// TIA Portal V20 export
TYPE "LBP_typeModularMcpModeGroupInput"
TITLE = Modular MCP image / Image MCP modulaire
// Input image of mode group keypad for modular MCP / Image des entrées du pupitre de groupes de modes de fonctionnement pour MCP modulaires
   STRUCT
      reset : Bool;   // input image n+0 bit 0 / Image des entrées n+0 bit 0
      cycleStop : Bool;   // input image n+0 bit 1 / Image des entrées n+0 bit 1
      cycleStart : Bool;   // input image n+0 bit 2 / Image des entrées n+0 bit 2
      singleBlock : Bool;   // input image n+0 bit 3 / Image des entrées n+0 bit 3
      inc100 : Bool;   // input image n+0 bit 4 / Image des entrées n+0 bit 4
      inc1000 : Bool;   // input image n+0 bit 5 / Image des entrées n+0 bit 5
      auto : Bool;   // input image n+0 bit 6 / Image des entrées n+0 bit 6
      inc1 : Bool;   // input image n+0 bit 7 / Image des entrées n+0 bit 7
      inc10 : Bool;   // input image n+1 bit 0 / Image des entrées n+1 bit 0
      mda : Bool;   // input image n+1 bit 1 / Image des entrées n+1 bit 1
      teachIn : Bool;   // input image n+1 bit 2 / Image des entrées n+1 bit 2
      incVar : Bool;   // input image n+1 bit 3 / Image des entrées n+1 bit 3
      jog : Bool;   // input image n+1 bit 4 / Image des entrées n+1 bit 4
      repos : Bool;   // input image n+1 bit 5 / Image des entrées n+1 bit 5
      refPoint : Bool;   // input image n+1 bit 6 / Image des entrées n+1 bit 6
      reserved17 : Bool;
      key16 : Bool;   // input image n+2 bit 0 / Image des entrées n+2 bit 0
      key17 : Bool;   // input image n+2 bit 1 / Image des entrées n+2 bit 1
      key18 : Bool;   // input image n+2 bit 2 / Image des entrées n+2 bit 2
      reserved23 : Bool;
      reserved24 : Bool;
      reserved25 : Bool;
      reserved26 : Bool;
      reserved27 : Bool;
      key24 : Bool;   // input image n+3 bit 0 / Image des entrées n+3 bit 0
      key25 : Bool;   // input image n+3 bit 1 / Image des entrées n+3 bit 1
      key26 : Bool;   // input image n+3 bit 2 / Image des entrées n+3 bit 2
      reserved33 : Bool;
      reserved34 : Bool;
      reserved35 : Bool;
      reserved36 : Bool;
      reserved37 : Bool;
   END_STRUCT;
END_TYPE
